// TwinCAT 3 PLC project Sample03
// ProgramVersion: 3.1.4020.1
// libraries:
//   Tc2_Standard, * (Beckhoff Automation GmbH)
//   Tc2_System, * (Beckhoff Automation GmbH)
//   Tc3_Module, * (Beckhoff Automation GmbH)
// project tree:
//   / PlcTask.TcTTO
//   POUs/ F_CalcSum3DimArray.TcPOU, MAIN.TcPOU
// real-time tasks:
//   TASK PlcTask: cycle T#10ms, priority 20, ADS port 350

CONFIGURATION Sample03
    RESOURCE PLC ON TwinCAT3
        TASK PlcTask(INTERVAL := T#10ms, PRIORITY := 20);
        PROGRAM MAIN WITH PlcTask : MAIN;
    END_RESOURCE
END_CONFIGURATION

// ---- POUs/MAIN.TcPOU
PROGRAM MAIN
VAR
	array01		: ARRAY[1..2, 3..4, 5..6] OF LREAL := [16.1, 34.1, 4.1, 43.1, 35.1, 2.1, 65.1, 16.1];
	lrSum01		: LREAL;
END_VAR

lrSum01 := F_CalcSum3DimArray(array01);

END_PROGRAM

// ---- POUs/F_CalcSum3DimArray.TcPOU
FUNCTION F_CalcSum3DimArray : LREAL
VAR_IN_OUT
	arrData		: ARRAY[*, *, *] OF LREAL;
END_VAR
VAR
	nIndex1, nIndex2, nIndex3	: DINT;
END_VAR

F_CalcSum3DimArray := 0;
FOR nIndex1 := LOWER_BOUND(arrData, 1) TO UPPER_BOUND(arrData, 1) DO
	FOR nIndex2 := LOWER_BOUND(arrData, 2) TO UPPER_BOUND(arrData, 2) DO
		FOR nIndex3 := LOWER_BOUND(arrData, 3) TO UPPER_BOUND(arrData, 3) DO
			F_CalcSum3DimArray := F_CalcSum3DimArray + arrData[nIndex1, nIndex2, nIndex3];
		END_FOR
	END_FOR
END_FOR

END_FUNCTION
